{attribute addProperty BoxType "EPP2816-0008-0016"}
{attribute addProperty Id "OutputAT %Q*ARRAY[0 ..7] OF BOOL6480"}
{attribute addProperty CRC "1062725746"}
{attribute addProperty SizeInBites "64"}
{attribute addProperty SizeInBytes "8"}
TYPE DIG_Outputs_Channel_33B76376 :
STRUCT
	{attribute addProperty Name "Output"}
	Output AT %Q* : ARRAY[0 ..7] OF BOOL;
END_STRUCT
END_TYPE

(* stored: Version 1.2.0.0, ProductVersion 3.1.4024.9
   DUT DIG_Outputs_Channel_33B76376: Id {b9376053-2c62-4a2a-af7d-c9e4ed11b908} *)
